(* PLC project Unnamed, Unknown Unnamed 1 *)
(* stored: creationDateTime 2026-03-24T09:46:09, modificationDateTime 2026-03-24T17:05:37 *)

PROGRAM program0
  VAR
    Start : BOOL;
    Stop : BOOL;
    RunState : BOOL;
    MRa : BOOL;
    MRb : BOOL;
    MLa : BOOL;
    MLb : BOOL;
    MUa : BOOL;
    MUb : BOOL;
    MCa : BOOL;
    MCb : BOOL;
    SR0 : SR;
    TP0 : TP;
    TP1 : TP;
    TP2 : TP;
    TP3 : TP;
    TP4 : TP;
    TP5 : TP;
    TP6 : TP;
    TP7 : TP;
    TP8 : TP;
  END_VAR

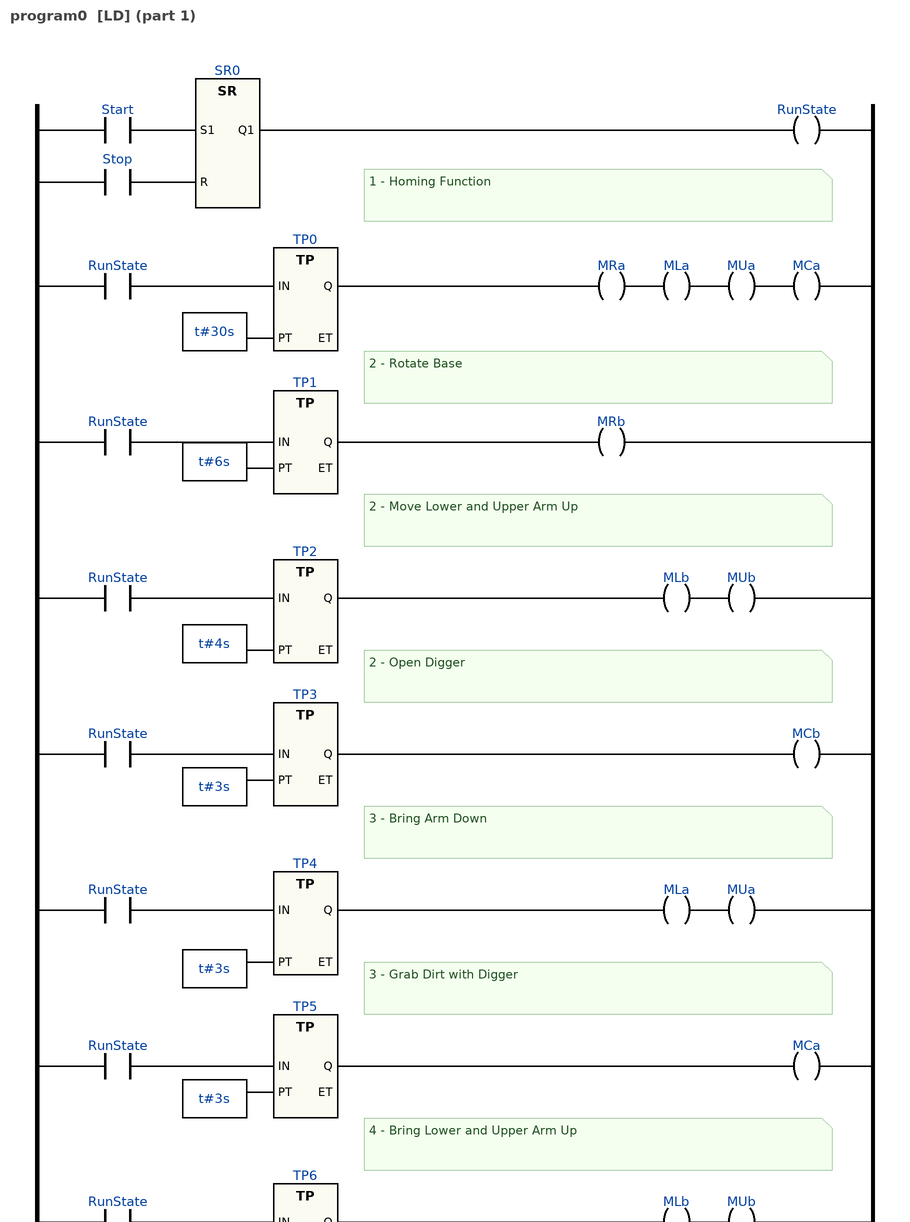
(* LD diagram, written out as Structured Text *)
SR0(S1 := Start, R := Stop);
RunState := SR0.Q1;
(* 1 - Homing Function *)
TP0(IN := RunState, PT := t#30s);
MCa := TP0.Q;
MLa := TP0.Q;
MRa := TP0.Q;
MUa := TP0.Q;
(* 2 - Rotate Base *)
TP1(IN := RunState, PT := t#6s);
MRb := TP1.Q;
(* 2 - Move Lower and Upper Arm Up *)
TP2(IN := RunState, PT := t#4s);
MLb := TP2.Q;
MUb := TP2.Q;
(* 2 - Open Digger *)
TP3(IN := RunState, PT := t#3s);
MCb := TP3.Q;
(* 3 - Bring Arm Down *)
TP4(IN := RunState, PT := t#3s);
MUa := TP4.Q;
MLa := TP4.Q;
(* 3 - Grab Dirt with Digger *)
TP5(IN := RunState, PT := t#3s);
MCa := TP5.Q;
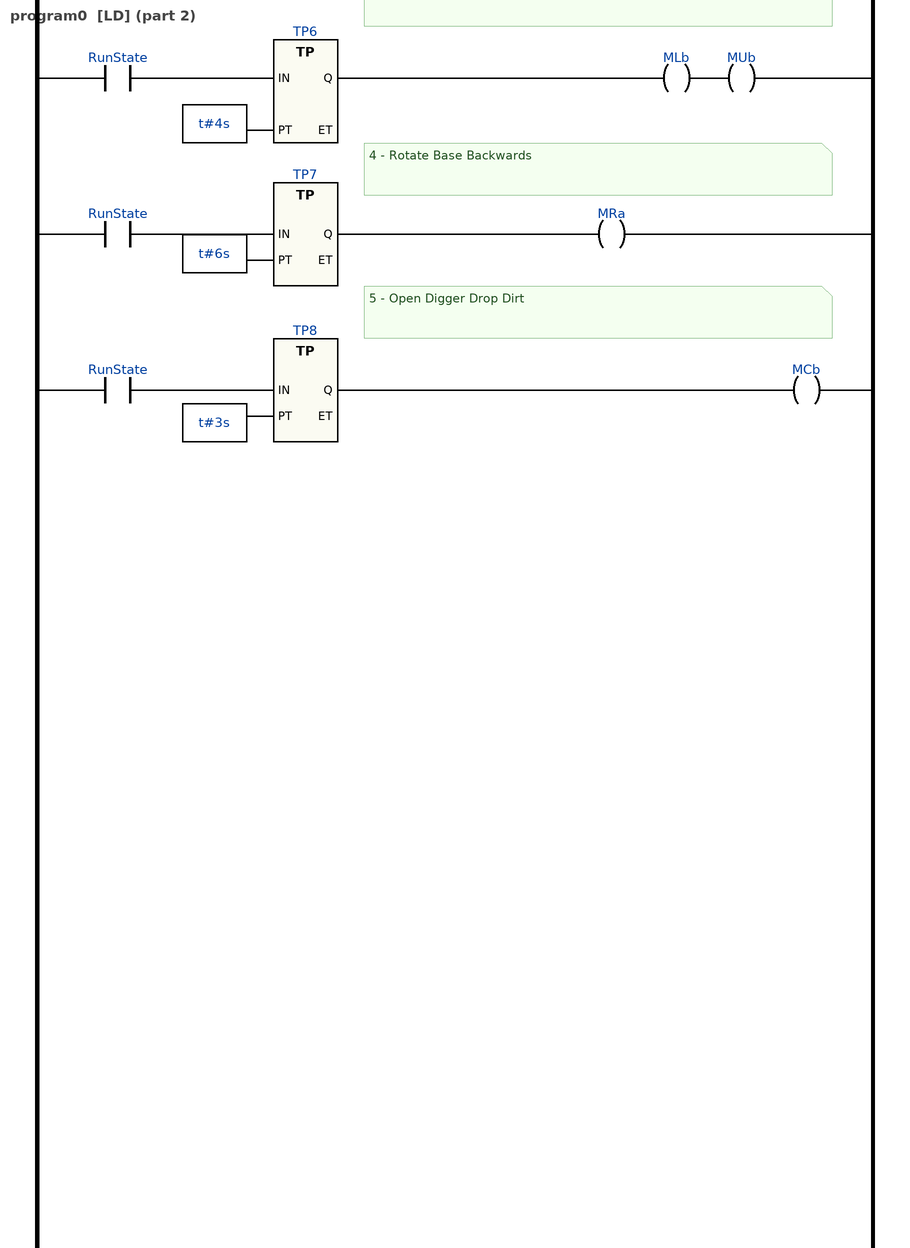
(* 4 - Bring Lower and Upper Arm Up *)
TP6(IN := RunState, PT := t#4s);
MUb := TP6.Q;
MLb := TP6.Q;
(* 4 - Rotate Base Backwards *)
TP7(IN := RunState, PT := t#6s);
MRa := TP7.Q;
(* 5 - Open Digger Drop Dirt *)
TP8(IN := RunState, PT := t#3s);
MCb := TP8.Q;
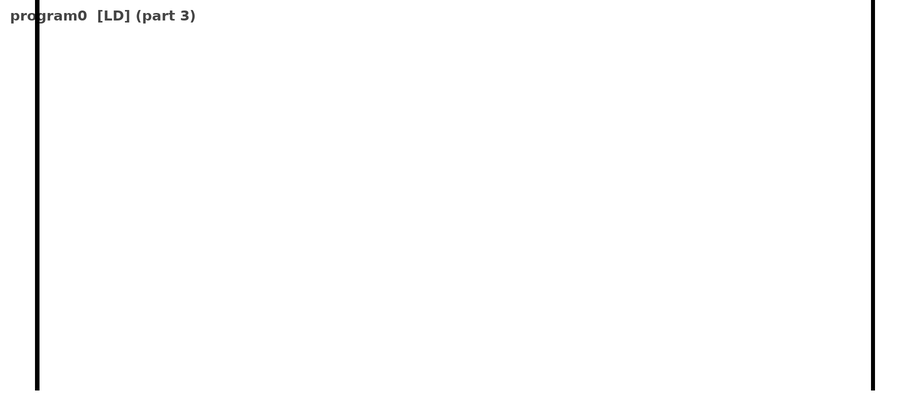
END_PROGRAM

CONFIGURATION Config0
  RESOURCE Res0 ON PLC
    TASK task0(INTERVAL := T#20ms, PRIORITY := 0);
    PROGRAM instance0 WITH task0 : program0;
  END_RESOURCE
END_CONFIGURATION
